FUNCTION_BLOCK T_ExternalControllerCollection EXTENDS T_CollectionBase

METHOD PUBLIC AddController : BOOL
VAR_INPUT
  newController : I_PackML_ExternalController;
END_VAR
VAR
	item : I_InterfaceBase;
END_VAR
IF newController = 0 THEN
	LogError( 'Cannot AddComponent invalid ref' );
	RETURN;
END_IF

IF NOT __QUERYINTERFACE(newController, item) THEN
	LogError( 'Cannot AddComponent  NOT __QUERYINTERFACE(newComponent, item)' );
	RETURN;
END_IF

IF HasItem( item := item ) THEN
	LogWarning( 'Component already in collection.' );
	RETURN;
END_IF

AddController := addInSpareSlot( item := item );
END_METHOD

METHOD PUBLIC ClearGroup // clears the group down
SUPER^.ClearGroup();
END_METHOD

METHOD PUBLIC NotifyModeChanged
VAR_INPUT
    Mode : E_PMLUnitMode;
END_VAR
VAR
	i : UDINT;
	Controller : I_PackML_ExternalController;
	item : I_InterfaceBase;
END_VAR
IF Count = 0 THEN
  RETURN;
END_IF

FOR i := 0 TO Count -1 DO

	IF NOT 	TryGetItem(i, item => item) THEN
		RETURN;
	END_IF
	
	IF NOT __QUERYINTERFACE(item, Controller) THEN
		RETURN;
	END_IF
		
	Controller.ModeChanged(Mode);
		
END_FOR
END_METHOD

METHOD PUBLIC NotifyStateChanged
VAR_INPUT
	CommandedState : Tc3_PackML_V2.E_PMLCommand;
END_VAR
VAR
	i : UDINT;
	Controller : I_PackML_ExternalController;
	item : I_InterfaceBase;
END_VAR
IF Count = 0 THEN
  RETURN;
END_IF

FOR i := 0 TO Count -1 DO

	IF NOT 	TryGetItem(i, item => item) THEN
		RETURN;
	END_IF
	
	IF NOT __QUERYINTERFACE(item, Controller) THEN
		RETURN;
	END_IF
		
	Controller.StateChanged(CommandedState);
		
END_FOR
END_METHOD

METHOD TryGetController: BOOL
VAR_INPUT
	index : UDINT;
END_VAR
VAR_OUTPUT
	Controller : I_PackML_ExternalController;
END_VAR
VAR
	item : I_InterfaceBase;
END_VAR
IF NOT SUPER^.TryGetItem(index := index, item => item) THEN
	LogError( 'Cannot TryGetComponent NOT SUPER^.TryGetItem(index := index, item => item) ' );
	RETURN;
END_IF

IF NOT __QUERYINTERFACE(item, Controller) THEN
	LogError( 'Cannot TryGetComponent   NOT __QUERYINTERFACE(item, component) ' );
	RETURN;
END_IF

TryGetController := Controller <> 0;
END_METHOD

END_FUNCTION_BLOCK

(* stored: Version 1.1.0.1, ProductVersion 3.1.4024.12
   POU T_ExternalControllerCollection: Id {c5e8f026-4eab-44f0-ace5-27f246664882}, SpecialFunc None
   Method AddController: Id {35a6c324-9983-499e-b12d-516396eb1406}
   Method ClearGroup: Id {054439b6-c605-4a05-bfee-f8050dc694af}
   Method NotifyModeChanged: Id {17f6e3c4-7a01-4c8b-b055-d636340e3bb7}
   Method NotifyStateChanged: Id {eea1ad95-9606-42e7-93a3-3c98612b2ba8}
   Method TryGetController: Id {799866d3-5fcb-43cf-b544-809f9053e66f} *)
